FUNCTION_BLOCK FB_StopBlade
VAR_INPUT
	TENERPIEZA: BOOL;
END_VAR
VAR_OUTPUT
	ESTOYBLOQUEANDO: BOOL;
	STOPBLADE: BOOL;
END_VAR
VAR
	CSTOPBLADE: STOPBLADE := STOPBLADE_REPOSO;

END_VAR

(* El StopBlade está en estado de reposo hasta recibir instrucciones *)
IF TENERPIEZA THEN
		STOPBLADE := TENERPIEZA;
		ESTOYBLOQUEANDO:= TENERPIEZA;
ELSE
		STOPBLADE := TENERPIEZA;
		ESTOYBLOQUEANDO:= TENERPIEZA;
END_IF

END_FUNCTION_BLOCK

(* stored: Version 1.1.0.1, ProductVersion 3.1.4024.12
   POU FB_StopBlade: Id {a18bfb3f-97bd-4ce8-b578-438b54d71bcf}, SpecialFunc None *)
